TEXTLIST TextList_MU_state
  0 = 'off'
  1 = 'idle'
  2 = 'swapping'
  100 = 'error'
   = ''
END_TEXTLIST

(* stored: Version 1.1.0.1, ProductVersion 3.1.4024.11
   TextList TextList_MU_state: Id {0b06baa3-0548-4137-9c13-d96c0a4594e1} *)
